Staubli VAL3: exceptionHandle.dtx

mdesc mNomSpeed
public num nForceThreshold[6]
public num nSpeedThreshold[6]
public num nRosFlagCmd
